// TIA Portal V19 export
FUNCTION_BLOCK "LAxisCtrlApcFr_UnpubMC_Interpolate"   // FB19523, LAD
{ S7_Optimized_Access := 'TRUE' }
// stored: IsIECCheckEnabled true, MemoryReserve 100, SetENOAutomatically true
   VAR_INPUT
      cam { ExternalAccessible := 'False'; ExternalVisible := 'False'; ExternalWritable := 'False'} : DB_ANY;
      execute { ExternalAccessible := 'False'; ExternalVisible := 'False'; ExternalWritable := 'False'} : Bool;
   END_VAR
   VAR_OUTPUT
      done : Bool;
      busy : Bool;
      error { ExternalAccessible := 'False'; ExternalVisible := 'False'; ExternalWritable := 'False'} : Bool;
      errorID { ExternalAccessible := 'False'; ExternalVisible := 'False'; ExternalWritable := 'False'} : Word;
   END_VAR
   VAR
      statExecuteOld { ExternalAccessible := 'False'; ExternalVisible := 'False'; ExternalWritable := 'False'} : Bool;
      statCam { ExternalAccessible := 'False'; ExternalVisible := 'False'; ExternalWritable := 'False'} : DB_ANY;
      statCamType { ExternalAccessible := 'False'; ExternalVisible := 'False'; ExternalWritable := 'False'} : Int;
      instMC { ExternalAccessible := 'False'; ExternalVisible := 'False'; ExternalWritable := 'False'} : MC_INTERPOLATECAM;
   END_VAR
   VAR CONSTANT
      CAM_1K : Int := 1;
      CAM_10K : Int := 2;
      INVALID_CAM : Int := -3;
      IDLE : Int := 0;
      ERROR_INVALID_TECHNOLOGY_OBJECT : Word := 16#8002;
   END_VAR
BEGIN

REGION Network 1 (SCL)
   REGION EXECUTE
       IF #execute AND NOT #statExecuteOld THEN

           CASE TypeOfDB(#cam) OF
               TO_Cam:
                   #statCam := #cam;
                   #statCamType := #CAM_1K;

               TO_Cam_10k:
                   #statCam := #cam;
                   #statCamType := #CAM_10K;

               ELSE
                   #statCam := 0;
                   #statCamType := #INVALID_CAM;
           END_CASE;

       ELSIF NOT #execute AND (#statCamType < #IDLE) THEN
           #statCamType := #IDLE;

           // Outputs
           #error := FALSE;
           #errorID := 16#0000;
       END_IF;
   END_REGION

   // Edge detection
   #statExecuteOld := #execute;

   CASE #statCamType OF
       #IDLE:
           ;

       #CAM_1K,
       #CAM_10K:
           REGION VALID_CAM
               // Inputs 
               #instMC.Execute := #execute;

               CASE #statCamType OF
                   #CAM_1K:
                       "LAxisCtrlApcFr_UnpubMC_Interpolate1k"(cam:=#statCam,
                                                              instMC:=#instMC);

                   #CAM_10K:
                       "LAxisCtrlApcFr_UnpubMC_Interpolate10k"(cam:=#statCam,
                                                               instMC:=#instMC);

               END_CASE;

               // Outputs
               #done := #instMC.Done;
               #busy := #instMC.Busy;
               #error := #instMC.Error;
               #errorID := #instMC.ErrorId;


               // Status of MC instruction
               IF NOT #instMC.Busy
                   AND NOT #instMC.Done
                   AND NOT #instMC.Error
               THEN
                   // Not active
                   #statCamType := #IDLE;
               END_IF;
           END_REGION

       ELSE
           REGION INVALID_TECHNOLOGY_OBJECT
               // Outputs
               #error := TRUE;
               #errorID := #ERROR_INVALID_TECHNOLOGY_OBJECT;
           END_REGION
   END_CASE;
END_REGION
END_FUNCTION_BLOCK
